KUKA KRL program: PickPlaceSubroutinesBase.SRC, PickPlaceSubroutinesBase.DAT

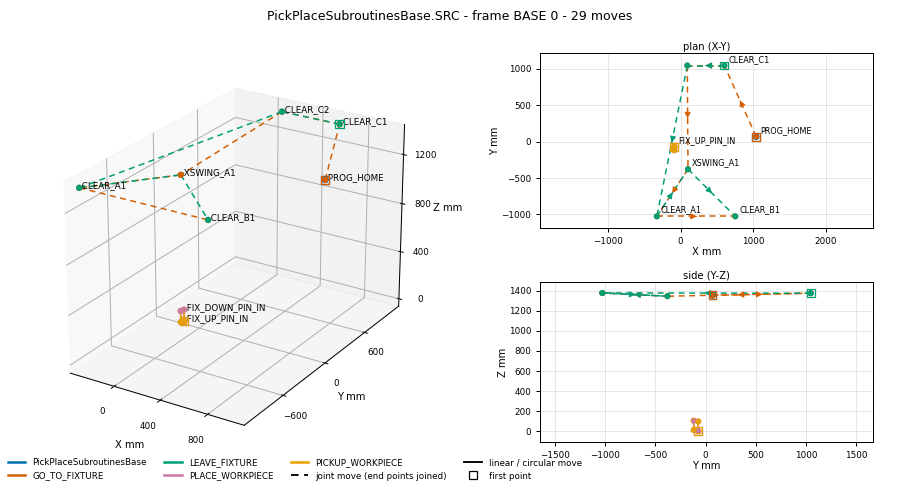
[picture p0: tool path of PickPlaceSubroutinesBase.SRC in frame BASE 0, 29 of 29 moves have a stored position in this frame; points joined in program order, loops and branches not executed]
--- PickPlaceSubroutinesBase.SRC ---
&ACCESS RVP1
&REL 10
&PARAM DISKPATH = KRC:\R1\Program
DEF PickPlaceSubroutinesBase()

; Declaration of KRL variables
DECL INT ret   ; Return value for RSI commands
DECL INT CONTID   ; ContainerID
DECL INT i
DECL INT j
DECL BOOL useRSI ; Do we use RSI
ENUM FIXTURE_ID A1, B1, C1, C2
ENUM FIXTURE_OPCODE PICK, PLACE

;FOLD INI
  ;FOLD BASISTECH INI
    GLOBAL INTERRUPT DECL 3 WHEN $STOPMESS==TRUE DO IR_STOPM ( )
    INTERRUPT ON 3
    BAS (#INITMOV,0 )
  ;ENDFOLD (BASISTECH INI)
  ;FOLD VEO INI

  ;ENDFOLD (VEO INI)
;ENDFOLD (INI)

;FOLD Joint Move Home
$BWDSTART=FALSE
PDAT_ACT=P2P_FULL_SPEED
FDAT_ACT=WORLD_FRAME
BAS(#PTP_PARAMS,100)
PTP PROG_HOME
;ENDFOLD

;FOLD Setup RSI
useRSI=TRUE
IF useRSI==TRUE THEN

  ; Create RSI Context
  ret = RSI_CREATE("RSI_Ethernet.rsi",CONTID,TRUE)
  IF (ret <> RSIOK) THEN
    HALT
  ENDIF

  ; Start RSI execution
  ret = RSI_ON(#RELATIVE)
  IF (ret <> RSIOK) THEN
    HALT
  ENDIF

ENDIF
;ENDFOLD

WAIT SEC 0.5; PAUSE TO REGISTER AT HOME

;FOLD WAIT FOR ( IN 1 'Button1' );%{PE}%R 8.3.41,%MKUKATPBASIS,%CEXT_WAIT_FOR,%VEXT_WAIT_FOR,%P 2:, 4:, 5:$IN, 6:1, 7:Button1, 9:
WAIT FOR  ( $IN[1] )
;ENDFOLD

FIXTURE_OP(#PICK, #C1)
FIXTURE_OP(#PLACE, #B1)
FIXTURE_OP(#PICK, #C2)
FIXTURE_OP(#PLACE, #A1)
;FOLD Joint Move Home
$BWDSTART=FALSE
PDAT_ACT=P2P_FULL_SPEED
FDAT_ACT=WORLD_FRAME
BAS(#PTP_PARAMS,100)
PTP PROG_HOME
;ENDFOLD

LOOP

;FOLD Wait for B1 Operator Finished
WAIT FOR  ( $IN[1] )
;ENDFOLD

FIXTURE_OP(#PICK, #B1)
FIXTURE_OP(#PLACE, #C1)
;FOLD Joint Move Home
$BWDSTART=FALSE
PDAT_ACT=P2P_FULL_SPEED
FDAT_ACT=WORLD_FRAME
BAS(#PTP_PARAMS,100)
PTP PROG_HOME
;ENDFOLD
FIXTURE_OP(#PICK, #C1)
FIXTURE_OP(#PLACE, #B1)
;FOLD Joint Move Home
$BWDSTART=FALSE
PDAT_ACT=P2P_FULL_SPEED
FDAT_ACT=WORLD_FRAME
BAS(#PTP_PARAMS,100)
PTP PROG_HOME
;ENDFOLD

;FOLD Wait for A1 Operator Finished
WAIT FOR  ( $IN[2] )
;ENDFOLD

FIXTURE_OP(#PICK, #A1)
FIXTURE_OP(#PLACE, #C2)
;FOLD Joint Move Home
$BWDSTART=FALSE
PDAT_ACT=P2P_FULL_SPEED
FDAT_ACT=WORLD_FRAME
BAS(#PTP_PARAMS,100)
PTP PROG_HOME
;ENDFOLD
FIXTURE_OP(#PICK, #C2)
FIXTURE_OP(#PLACE, #A1)
;FOLD Joint Move Home
$BWDSTART=FALSE
PDAT_ACT=P2P_FULL_SPEED
FDAT_ACT=WORLD_FRAME
BAS(#PTP_PARAMS,100)
PTP PROG_HOME
;ENDFOLD

ENDLOOP
END

DEF SET_SOLENOID_EXTEND(EXTENDED:IN)
  DECL BOOL EXTENDED
  $OUT[SOLENOID_ON_CHAN]=EXTENDED
  $OUT[SOLENOID_OFF_CHAN]=NOT EXTENDED
  $OUT[END_EFFECTOR_SIGNAL_CHAN]=EXTENDED
  RETURN
END

DEF EXTEND_SOLENOID()
  SET_SOLENOID_EXTEND(TRUE)
  RETURN
END

DEF RETRACT_SOLENOID()
  SET_SOLENOID_EXTEND(FALSE)
  RETURN
END

DEFFCT FDAT FRAME_FROM_FIXTURE(FIX_ID:IN)
  DECL FIXTURE_ID FIX_ID
  DECL FDAT RET_VAL
  SWITCH FIX_ID
    CASE #C1
      RET_VAL=FIXTURE_C1_FRAME
    CASE #C2
      RET_VAL=FIXTURE_C2_FRAME
    CASE #A1
      RET_VAL=FIXTURE_A_FRAME
    CASE #B1
      RET_VAL=FIXTURE_B_FRAME
    DEFAULT
      RET_VAL=WORLD_FRAME
      HALT
  ENDSWITCH
  RETURN RET_VAL
ENDFCT

DEF FIXTURE_OP(OPCODE:IN, FIX_ID:IN)
  DECL FIXTURE_ID FIX_ID
  DECL FIXTURE_OPCODE OPCODE
  DECL FDAT FIX_FRAME
  FIX_FRAME=FRAME_FROM_FIXTURE(FIX_ID)


  GO_TO_FIXTURE(FIX_ID)
  SWITCH OPCODE
    CASE #PICK
      PICKUP_WORKPIECE(FIX_FRAME)
    CASE #PLACE
      PLACE_WORKPIECE(FIX_FRAME)
    DEFAULT
    HALT
  ENDSWITCH
  LEAVE_FIXTURE(FIX_ID)
END

DEF GO_TO_FIXTURE(FIX_ID:IN)
  DECL FIXTURE_ID FIX_ID

  ;FOLD Approx Joint Move Home
  $BWDSTART=FALSE
  PDAT_ACT=P2P_FULL_SPEED
  FDAT_ACT=WORLD_FRAME
  BAS(#PTP_PARAMS,100)
  PTP PROG_HOME C_PTP
  ;ENDFOLD

  SWITCH FIX_ID
    CASE #C1
      ;FOLD PTP Clear C1
      $BWDSTART=FALSE
      PDAT_ACT=P2P_FULL_SPEED
      FDAT_ACT=WORLD_FRAME
      BAS(#PTP_PARAMS,100)
      PTP CLEAR_C1
      ;ENDFOLD
    CASE #C2
      ;FOLD PTP Clear C2
      $BWDSTART=FALSE
      PDAT_ACT=P2P_FULL_SPEED
      FDAT_ACT=WORLD_FRAME
      BAS(#PTP_PARAMS,100)
      PTP CLEAR_C2
      ;ENDFOLD
    CASE #A1
      ;FOLD PTP Swing A1
      $BWDSTART=FALSE
      PDAT_ACT=P2P_FULL_SPEED
      FDAT_ACT=WORLD_FRAME
      BAS(#PTP_PARAMS,100)
      PTP XSWING_A1
      ;ENDFOLD
      ;FOLD PTP Clear A1
      $BWDSTART=FALSE
      PDAT_ACT=P2P_FULL_SPEED
      FDAT_ACT=WORLD_FRAME
      BAS(#PTP_PARAMS,100)
      PTP CLEAR_A1
      ;ENDFOLD
    CASE #B1
      ;FOLD PTP Clear B1
      $BWDSTART=FALSE
      PDAT_ACT=P2P_FULL_SPEED
      FDAT_ACT=WORLD_FRAME
      BAS(#PTP_PARAMS,100)
      PTP CLEAR_B1
      ;ENDFOLD
    DEFAULT
      HALT
  ENDSWITCH
  RETURN
END

DEF LEAVE_FIXTURE(FIX_ID:IN)
  DECL FIXTURE_ID FIX_ID

  SWITCH FIX_ID
    CASE #C1
      ;FOLD PTP Clear C1
      $BWDSTART=FALSE
      PDAT_ACT=P2P_FULL_SPEED
      FDAT_ACT=WORLD_FRAME
      BAS(#PTP_PARAMS,100)
      PTP CLEAR_C1
      ;ENDFOLD
    CASE #C2
      ;FOLD PTP Clear C2
      $BWDSTART=FALSE
      PDAT_ACT=P2P_FULL_SPEED
      FDAT_ACT=WORLD_FRAME
      BAS(#PTP_PARAMS,100)
      PTP CLEAR_C2
      ;ENDFOLD
    CASE #A1
      ;FOLD PTP Clear A1
      $BWDSTART=FALSE
      PDAT_ACT=P2P_FULL_SPEED
      FDAT_ACT=WORLD_FRAME
      BAS(#PTP_PARAMS,100)
      PTP CLEAR_A1
      ;ENDFOLD
      ;FOLD PTP Swing A1
      $BWDSTART=FALSE
      PDAT_ACT=P2P_FULL_SPEED
      FDAT_ACT=WORLD_FRAME
      BAS(#PTP_PARAMS,100)
      PTP XSWING_A1
      ;ENDFOLD
    CASE #B1
      ;FOLD PTP Clear B1
      $BWDSTART=FALSE
      PDAT_ACT=P2P_FULL_SPEED
      FDAT_ACT=WORLD_FRAME
      BAS(#PTP_PARAMS,100)
      PTP CLEAR_B1
      ;ENDFOLD
    DEFAULT
      HALT
  ENDSWITCH
  RETURN
END

DEF PLACE_WORKPIECE(FIX_FRAME:IN)
  DECL FDAT FIX_FRAME

  ;FOLD Joint Move to Above
  $BWDSTART=FALSE
  PDAT_ACT=P2P_FULL_SPEED
  FDAT_ACT=FIX_FRAME
  BAS(#PTP_PARAMS,100)
  PTP FIX_UP_PIN_IN
  ;ENDFOLD
  ;FOLD Move to Above
  $BWDSTART=FALSE
  LDAT_ACT=LIN_TWO_MPS
  FDAT_ACT=FIX_FRAME
  BAS(#CP_PARAMS,2)
  LIN FIX_UP_PIN_IN
  ;ENDFOLD

  ;FOLD Drop part to fixture
  $BWDSTART=FALSE
  LDAT_ACT=LIN_TWO_MPS
  FDAT_ACT=FIX_FRAME
  BAS(#CP_PARAMS,2)
  LIN FIX_DOWN_PIN_IN
  ;ENDFOLD

  ;FOLD Release Part
  RETRACT_SOLENOID()
  WAIT SEC 0.75
  ;ENDFOLD

  ;FOLD Slide Pin Out
  $BWDSTART=FALSE
  LDAT_ACT=LIN_TWO_MPS
  FDAT_ACT=FIX_FRAME
  BAS(#CP_PARAMS,2)
  LIN FIX_DOWN_PIN_OUT
  ;ENDFOLD

  ;FOLD Pull up without part
  $BWDSTART=FALSE
  LDAT_ACT=LIN_TWO_MPS
  FDAT_ACT=FIX_FRAME
  BAS(#CP_PARAMS,2)
  LIN FIX_UP_PIN_OUT
  ;ENDFOLD

  ;FOLD Move to Above
  $BWDSTART=FALSE
  LDAT_ACT=LIN_TWO_MPS
  FDAT_ACT=FIX_FRAME
  BAS(#CP_PARAMS,2)
  LIN FIX_UP_PIN_IN
  ;ENDFOLD
END

DEF PICKUP_WORKPIECE(FIX_FRAME:IN)
  DECL FDAT FIX_FRAME

  ;FOLD Joint Move to Above
  $BWDSTART=FALSE
  PDAT_ACT=P2P_FULL_SPEED
  FDAT_ACT=FIX_FRAME
  BAS(#PTP_PARAMS,100)
  PTP FIX_UP_PIN_IN
  ;ENDFOLD
  ;FOLD Move to Above
  $BWDSTART=FALSE
  LDAT_ACT=LIN_TWO_MPS
  FDAT_ACT=FIX_FRAME
  BAS(#CP_PARAMS,2)
  LIN FIX_UP_PIN_IN
  ;ENDFOLD

  ;FOLD Move over to clear pin
  $BWDSTART=FALSE
  LDAT_ACT=LIN_TWO_MPS
  FDAT_ACT=FIX_FRAME
  BAS(#CP_PARAMS,2)
  LIN FIX_UP_PIN_OUT
  ;ENDFOLD

  ;FOLD Drop down
  $BWDSTART=FALSE
  LDAT_ACT=LIN_TWO_MPS
  FDAT_ACT=FIX_FRAME
  BAS(#CP_PARAMS,2)
  LIN FIX_DOWN_PIN_OUT
  ;ENDFOLD

  ;FOLD Slide Pin In
  $BWDSTART=FALSE
  LDAT_ACT=LIN_TWO_MPS
  FDAT_ACT=FIX_FRAME
  BAS(#CP_PARAMS,2)
  LIN FIX_DOWN_PIN_IN
  ;ENDFOLD

  ;FOLD Grab Part
  EXTEND_SOLENOID()
  WAIT SEC 0.75
  ;ENDFOLD

  ;FOLD Lift with Part
  $BWDSTART=FALSE
  LDAT_ACT=LIN_TWO_MPS
  FDAT_ACT=FIX_FRAME
  BAS(#CP_PARAMS,2)
  LIN FIX_UP_PIN_IN
  ;ENDFOLD
END

--- PickPlaceSubroutinesBase.DAT ---
&ACCESS RVP1
&REL 10
&PARAM DISKPATH = KRC:\R1\Program
DEFDAT  PickPlaceSubroutinesBase PUBLIC
;FOLD EXTERNAL DECLARATIONS;%{PE}%MKUKATPBASIS,%CEXT,%VCOMMON,%P
;FOLD BASISTECH EXT;%{PE}%MKUKATPBASIS,%CEXT,%VEXT,%P
EXT  BAS (BAS_COMMAND  :IN,REAL  :IN )
DECL INT SUCCESS
;ENDFOLD (BASISTECH EXT)

;FOLD VEO EXT;%{E}%MKUKATPUSER,%CEXT,%VEXT,%P
DECL INT SOLENOID_ON_CHAN=2
DECL INT SOLENOID_OFF_CHAN=3
DECL INT END_EFFECTOR_SIGNAL_CHAN=1

;ENDFOLD (VEO EXT)
;ENDFOLD (EXTERNAL DECLARATIONS)

;DECL BASIS_SUGG_T LAST_BASIS={POINT1[] "CLEAR_B1                ",POINT2[] "CLEAR_B1                ",CP_PARAMS[] "CPDAT19                 ",PTP_PARAMS[] "PDAT32                  ",CONT[] "                        ",CP_VEL[] "2                       ",PTP_VEL[] "100                     ",SYNC_PARAMS[] "SYNCDAT                 ",SPL_NAME[] "S0                      ",A_PARAMS[] "ADAT0                   "}

; Motion Params
DECL PDAT P2P_FULL_SPEED={VEL 100.000,ACC 100.000,APO_DIST 100.000,GEAR_JERK 50.0000,EXAX_IGN 0}
DECL LDAT LIN_TWO_MPS={VEL 2.00000,ACC 100.000,APO_DIST 100.000,APO_FAC 50.0000,AXIS_VEL 100.000,AXIS_ACC 100.000,ORI_TYP #VAR,CIRC_TYP #BASE,JERK_FAC 50.0000,GEAR_JERK 50.0000,EXAX_IGN 0}

; Motion Frames
DECL GLOBAL CONST FDAT WORLD_FRAME={TOOL_NO 0,BASE_NO 0,IPO_FRAME #BASE,POINT2[] " ",TQ_STATE FALSE}
DECL GLOBAL CONST FDAT FIXTURE_A_FRAME={TOOL_NO 2,BASE_NO 1,IPO_FRAME #BASE,POINT2[] " ",TQ_STATE FALSE}
DECL GLOBAL CONST FDAT FIXTURE_B_FRAME={TOOL_NO 2,BASE_NO 2,IPO_FRAME #BASE,POINT2[] " ",TQ_STATE FALSE}
DECL GLOBAL CONST FDAT FIXTURE_C1_FRAME={TOOL_NO 2,BASE_NO 3,IPO_FRAME #BASE,POINT2[] " ",TQ_STATE FALSE}
DECL GLOBAL CONST FDAT FIXTURE_C2_FRAME={TOOL_NO 2,BASE_NO 4,IPO_FRAME #BASE,POINT2[] " ",TQ_STATE FALSE}

; Home
DECL CONST POS PROG_HOME={X 1038.76978,Y 69.6914444,Z 1353.78125,A 90.5040741,B 1.11831033,C 101.029724,S 2,T 35}

; Above Fixture C1
DECL CONST POS ABOVE_C1={X 696.051,Y 1160.38928,Z 1264.14661,A 88.3531342,B -2.00895047,C 179.443344,S 2,T 43}
; Clear Fixture C1
DECL CONST POS CLEAR_C1={X 601.471375,Y 1046.63330,Z 1374.83582,A 141.312286,B -9.11080170,C 131.767487,S 2,T 35}

; Above Fixture C2
DECL CONST POS ABOVE_C2={X 196.378,Y 1160.51672,Z 1261.58508,A 88.8925247,B -0.838449419,C -178.863846,S 2,T 43}
; Clear Fixture C2
DECL CONST POS CLEAR_C2={X 91.9833374,Y 1046.63330,Z 1374.83582,A 141.312286,B -9.11080170,C 131.767487,S 2,T 35}

; Above Fixture A1
DECL CONST POS ABOVE_A1={X -289.070984,Y -1087.14709,Z 1307.36121,A 93.9495621,B -0.198399931,C 179.599365,S 2,T 10}
; Clear Fixture A1
DECL CONST POS CLEAR_A1={X -327.022125,Y -1026.90161,Z 1377.38989,A 87.8513184,B 21.0648441,C -172.710373,S 2,T 2}
; Swing in while moving toward A1 to clear B1
DECL CONST POS XSWING_A1={X 101.377792,Y -378.924896,Z 1344.78638,A 29.9830952,B 19.5461426,C 115.466858,S 2,T 42}

; Above Fixture B1
DECL CONST POS ABOVE_B1={X 764.500244,Y -1109.62524,Z 1310.77991,A 89.1244125,B -0.197261065,C 179.599319,S 2,T 42}
; Clear Fixture B1
DECL CONST POS CLEAR_B1={X 751.899048,Y -1026.90076,Z 1377.38928,A 87.8513107,B 21.0648422,C -172.710388,S 2,T 34}

; Pick / Place Base Relative Linear Moves
DECL CONST POS FIX_UP_PIN_IN={X -87.3149338,Y -71.6395,Z 1.23888421,A -0.000531545433,B -0.00384448632,C -99.0039291}
DECL CONST POS FIX_DOWN_PIN_IN={X -88.1166382,Y -71.9804840,Z 98.6590118,A -0.000532631762,B -0.00384636899,C -99.0039291}
DECL CONST POS FIX_DOWN_PIN_OUT={X -88.1176071,Y -117.477814,Z 105.868248,A -0.000533006387,B -0.00384651637,C -99.0039291}
DECL CONST POS FIX_UP_PIN_OUT={X -87.3406601,Y -117.154099,Z 13.1294451,A -0.000533087587,B -0.00384653918,C -99.0039291}

; Place Relative Linear Moves
DECL CONST POS PLACE_DOWN_PIN_IN={Z -120.040894}
DECL CONST POS PLACE_DOWN_PIN_OUT={X -43.5248413,Y 0.690670,Z -7.42041}
DECL CONST POS PLACE_UP_PIN_OUT={Y -1.00000E-04,Z 87.0101318}
DECL CONST POS PLACE_ABOVE_WITHOUT_PART={X 43.5247803,Y -0.690550,Z 40.4511719}

; Pick Relative Linear Moves
DECL CONST POS PICK_UP_PIN_OUT={X -43.5247803,Y 0.690550,Z -40.4511719}
DECL CONST POS PICK_DOWN_PIN_OUT={Z -87.0101318}
DECL CONST POS PICK_DOWN_PIN_IN={X 43.5248413,Y -0.690670,Z 7.42041}
DECL CONST POS PICK_UP_WITH_PART={Z 120.040894}

ENDDAT
